FUNCTION_BLOCK SWITCH3 (* Basic function block for Demux 3 events *)
  (* Standard: 61499-2; Classification: EventProcessing; ApplicationDomain: Modelling and Processing *)
  (* Version 1.0, 2018-05-29, Duc Do Tran, OFFIS e.V. *)
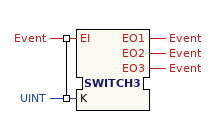
  EVENT_INPUT
    EI WITH K;
  END_EVENT
  EVENT_OUTPUT
    EO1;
    EO2;
    EO3;
  END_EVENT
  VAR_INPUT
    K : UINT;
  END_VAR
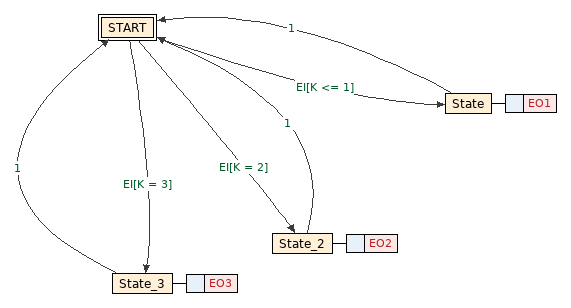
  EC_STATES
    START; (* Initial State *)
    State : -> EO1;
    State_2 : -> EO2;
    State_3 : -> EO3;
  END_STATES
  EC_TRANSITIONS
    START TO State := EI[K <= 1];
    State TO START := 1;
    START TO State_2 := EI[K = 2];
    START TO State_3 := EI[K = 3];
    State_3 TO START := 1;
    State_2 TO START := 1;
  END_TRANSITIONS
END_FUNCTION_BLOCK
